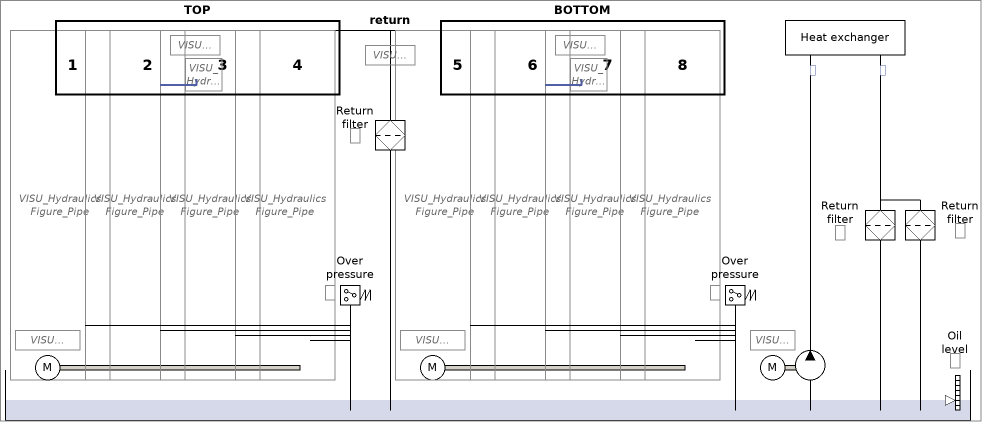
VISUALIZATION VISU_HydraulicsFigure  // 982x422
VAR_IN_OUT
    ref : Hydraulics;
    widget : HydraulicsWidget;
	ref_safety : SafetyHydraulics;
END_VAR
    Rectangle (775,365 35x5)
    Rectangle (440,365 245x5)
    Ellipse (420,355 25x25), "M"
    Rectangle (5,400 965x20)
    Rectangle (55,365 245x5)
    Line (5,370) (5,420)
    Line (5,420) (970,420)
    Line (85,30) (695,30)
    Frame (10,30 100x350)
        shows VISU_HydraulicsFigure_Pipe(underpressureOK := ref_safety.top1NoUnderpressure, filterOK := ref.parts.top.entranceFilter1OK)
    Frame (85,30 100x350)
        shows VISU_HydraulicsFigure_Pipe(underpressureOK := ref_safety.top2NoUnderpressure, filterOK := ref.parts.top.entranceFilter2OK)
    Frame (160,30 100x350)
        shows VISU_HydraulicsFigure_Pipe(underpressureOK := ref_safety.top3NoUnderpressure, filterOK := ref.parts.top.entranceFilter3OK)
    Frame (235,30 100x350)
        shows VISU_HydraulicsFigure_Pipe(underpressureOK := ref_safety.top4NoUnderpressure, filterOK := ref.parts.top.entranceFilter4OK)
    Frame (395,30 100x350)
        shows VISU_HydraulicsFigure_Pipe(underpressureOK := ref_safety.bottom5NoUnderpressure, filterOK := ref.parts.bottom.entranceFilter1OK)
    Frame (470,30 100x350)
        shows VISU_HydraulicsFigure_Pipe(underpressureOK := ref_safety.bottom6NoUnderpressure, filterOK := ref.parts.bottom.entranceFilter2OK)
    Frame (545,30 100x350)
        shows VISU_HydraulicsFigure_Pipe(underpressureOK := ref_safety.bottom7NoUnderpressure, filterOK := ref.parts.bottom.entranceFilter3OK)
    Frame (620,30 100x350)
        shows VISU_HydraulicsFigure_Pipe(underpressureOK := ref_safety.bottom8NoUnderpressure, filterOK := ref.parts.bottom.entranceFilter4OK)
    Line (85,325) (350,325)
    Line (160,330) (350,330)
    Line (235,335) (350,335)
    Line (310,340) (350,340)
    Line (350,305) (350,410)
    Line (390,30) (390,410)
    Line (970,370) (970,420)
    Rectangle (340,285 20x20)
    Polyline (360,300) (365,290) (365,300) (370,290) (370,300)
    Line (345,290) (355,295)
    Ellipse (344,289 4x4)
    Ellipse (344,297 4x4)
    Ellipse (352,293 4x4)
    Frame (325,285 10x15)
        shows VISU_State_red_green(state := ref_safety.topNoOverpressure)
    Label (320,250 60x35), "Over pressure"
    Line (470,325) (735,325)
    Line (545,330) (735,330)
    Line (620,335) (735,335)
    Line (695,340) (735,340)
    Line (735,305) (735,410)
    Rectangle (725,285 20x20)
    Polyline (745,300) (750,290) (750,300) (755,290) (755,300)
    Line (730,290) (740,295)
    Ellipse (729,289 4x4)
    Ellipse (729,297 4x4)
    Ellipse (737,293 4x4)
    Frame (710,285 10x15)
        shows VISU_State_red_green(state := ref_safety.bottomNoOverpressure)
    Label (705,250 60x35), "Over pressure"
    Ellipse (35,355 25x25), "M"
    RoundedRectangle (440,20 285x75)
    Label (440,0 285x20), "BOTTOM"
    Label (55,0 285x20), "TOP"
    RoundedRectangle (55,20 285x75)
    Frame (15,330 65x20)
        shows VISU_StatusWidget(widget := widget.top.driveStatus)
    Frame (400,330 65x20)
        shows VISU_StatusWidget(widget := widget.bottom.driveStatus)
    Label (65,55 15x20), "1"
    Label (140,55 15x20), "2"
    Label (215,55 15x20), "3"
    Label (290,55 15x20), "4"
    Label (450,55 15x20), "5"
    Label (525,55 15x20), "6"
    Label (600,55 15x20), "7"
    Label (675,55 15x20), "8"
    Frame (185,58 37x33)
        shows VISU_HydraulicsFigure_Manometer()
    Polyline (196,79) (196,85) (160,85)
    Frame (170,35 50x20)
        shows VISU_StatusWidget(widget := widget.top.pressureStatus)
    Frame (555,35 50x20)
        shows VISU_StatusWidget(widget := widget.bottom.pressureStatus)
    Frame (570,58 37x33)
        shows VISU_HydraulicsFigure_Manometer()
    Polyline (581,79) (581,85) (545,85)
    Frame (365,45 50x20)
        shows VISU_StatusWidget(widget := widget.bearingTemperatureStatus)
    Label (340,10 100x20), "return"
    Rectangle (375,120 30x30)
    Polygon (375,135) (390,120) (405,135) (390,150)
    Line (375,135) (380,135)
    Line (395,135) (400,135)
    Line (385,135) (390,135)
    Label (335,100 40x35), "Return filter"
    Frame (350,128 10x15)
        shows VISU_State_green_red(state := ref_safety.returnFilterOverpressure)
    Line (810,75) (810,350)
    Ellipse (795,350 30x30)
    Polygon (805,360) (810,350) (815,360)
    Line (810,380) (810,410)
    Rectangle (905,210 30x30)
    Polygon (905,225) (920,210) (935,225) (920,240)
    Line (905,225) (910,225)
    Line (925,225) (930,225)
    Line (915,225) (920,225)
    Label (940,195 40x35), "Return filter"
    Frame (955,223 10x15)
        shows VISU_State_red_green(state := ref.circulationFilterDOK)
    Rectangle (865,210 30x30)
    Polygon (865,225) (880,210) (895,225) (880,240)
    Line (865,225) (870,225)
    Line (885,225) (890,225)
    Line (875,225) (880,225)
    Label (820,195 40x35), "Return filter"
    Line (880,240) (880,410)
    Line (920,240) (920,410)
    Line (880,75) (880,210)
    Line (920,200) (920,210)
    Line (920,200) (880,200)
    Polygon (810,65) (815,65) (815,75) (810,75)
    Polygon (880,65) (885,65) (885,75) (880,75)
    Line (880,55) (880,65)
    Line (810,55) (810,65)
    Rectangle (785,20 120x35), "Heat exchanger"
    Ellipse (760,355 25x25), "M"
    Rectangle (955,375 5x35)
    Polygon (945,405) (945,395) (955,400)
    Line (955,380) (960,380)
    Line (955,385) (960,385)
    Line (955,390) (960,390)
    Line (955,395) (960,395)
    Line (955,400) (960,400)
    Line (955,405) (960,405)
    Frame (950,353 10x15)
        shows VISU_State_green_red(state := ref.oilLevelTooHigh)
    Label (935,325 40x35), "Oil level"
    Frame (835,225 10x15)
        shows VISU_State_red_green(state := ref.circulationFilterGOK)
    Frame (750,330 45x20)
        shows VISU_StatusWidget(widget := widget.circulationStatus)
END_VISUALIZATION

(* stored: Version 1.1.0.1, ProductVersion 3.1.4019.2
   Visu VISU_HydraulicsFigure: Id {3031a4d2-571a-484f-ba09-a12914b190fb} *)
